PROGRAM Main2
VAR
    nCounter: UINT;
END_VAR

nCounter := nCounter + 1;

END_PROGRAM

(* stored: Version 1.1.0.1
   POU Main2: Id {f196da23-5028-47d2-968c-46b028689f25}, SpecialFunc None *)
